(* IEC 61131-3 sources: CodesysTest/alpha/export/Device.dev/Plc Logic/Application/FBs/DataHandlers/FB_ModbusDWORD.pou/RawValue.prop, 1 file *)

(* ---- Set.pm.st ---- *)
(*#-#-#-#-#-#-#-#-#-#---Declaration---#-#-#-#-#-#-#-#-#-#-#-#-#*)

VAR
END_VAR
(*#-#-#-#-#-#-#-#-#-#---Implementation---#-#-#-#-#-#-#-#-#-#-#-#-#*)

_rawValue := RawValue;
_highWord := OSCAT_BASIC.WORD_OF_DWORD(in := _rawValue, N := 1);
_lowWord := OSCAT_BASIC.WORD_OF_DWORD(in := _rawValue, N := 0);
